PROGRAM POU_UserInterface
VAR
	inputSawingLength : INT;
	inputSawingSpeed: INT :=1;	//default value
	startButtonLengthStop: BOOL;
	messageMoveMetalToStop : BOOL;
	startClamp : BOOL;
	sawingDone: BOOL;
	timer1 : ton;
	
	
	signStartClamping: BOOL;
	timer1Start: BOOL;
	time1: TIME;
	timer1Reached: BOOL;
END_VAR

gvl.requiredSawingLength := inputSawingLength;
IF startButtonLengthStop THEN
	gvl.startButtonLengthStop := TRUE;
END_IF

IF gvl.stopPosReached and not gvl.metalIsToStop THEN
	gvl.startButtonLengthStop:= FALSE;
	messagemovemetaltostop := TRUE;
ELSE
		messagemovemetaltostop := FALSE;
END_IF

signStartClamping := gvl.metalIsToStop;
gvl.sawingSpeed := inputsawingspeed;

IF  startClamp THEN
	gvl.startClamp := TRUE;
	
END_IF

IF gvl.metalIsToStop THEN
	messagemovemetaltostop := FALSE; 
END_IF

IF gvl.sawingProcessDone THEN
	sawingDone :=TRUE;
	gvl.startClamp := FALSE;
	timer1Start := TRUE;
	time1 := T#3S;
END_IF

IF timer1reached THEN
	sawingdone:= FALSE;
	timer1start := FALSE;
END_IF

timer1(in:= timer1start, pt := time1, q => timer1reached);

END_PROGRAM

(* stored: Version 1.1.0.1, ProductVersion 3.1.4024.12
   POU POU_UserInterface: Id {84ac30c7-5aab-413f-8e32-caf8995e0e5a}, SpecialFunc None *)
